# EPICS autosave request: support/optics-2-7/opticsApp/Db/CoarseFineMotor_settings.req
$(P)MOT.TWV
$(P)mode
$(P)fineMode
